{attribute 'GeneratedUsingTerminal: EP9214-0023-0019'}
{attribute addProperty BoxType "EP9214-0023-0019"}
{attribute addProperty Id "Temperature_WarningAT %I*BOOL1Temperature_ErrorAT %I*BOOL1Us_WarningAT %I*BOOL1Us_ErrorAT %I*BOOL1Up_WarningAT %I*BOOL1Up_ErrorAT %I*BOOL1Global_Error_BitAT %I*BOOL1Reset_InputAT %I*BOOL1TxPDO_StateAT %I*BOOL1TxPDO_ToggleAT %I*BOOL1"}
{attribute addProperty CRC "2601048341"}
{attribute addProperty Size "10"}
TYPE DPO_Inputs_Device_9B08D915 :
STRUCT
	{attribute addProperty Name "Temperature_Warning"}
	Temperature_Warning AT %I* : BOOL;
	{attribute addProperty Name "Temperature_Error"}
	Temperature_Error AT %I* : BOOL;
	{attribute addProperty Name "Us_Warning"}
	Us_Warning AT %I* : BOOL;
	{attribute addProperty Name "Us_Error"}
	Us_Error AT %I* : BOOL;
	{attribute addProperty Name "Up_Warning"}
	Up_Warning AT %I* : BOOL;
	{attribute addProperty Name "Up_Error"}
	Up_Error AT %I* : BOOL;
	{attribute addProperty Name "Global_Error_Bit"}
	Global_Error_Bit AT %I* : BOOL;
	{attribute addProperty Name "Reset_Input"}
	Reset_Input AT %I* : BOOL;
	{attribute addProperty Name "TxPDO_State"}
	TxPDO_State AT %I* : BOOL;
	{attribute addProperty Name "TxPDO_Toggle"}
	TxPDO_Toggle AT %I* : BOOL;
END_STRUCT
END_TYPE

(* stored: Version 1.2.0.0, ProductVersion 3.1.4024.9
   DUT DPO_Inputs_Device_9B08D915: Id {0fcd4f7b-010e-4bd6-b457-83d29e14b925} *)
